PROGRAM ActuationSystems
VAR
fbMainJibCylinderHyd : ValveControlledCylinder;
fbKnuckleJibCylinderHyd : ValveControlledCylinder;
fbKingRotationCylinderHyd : ValveControlledCylinder;
//HydraulicCylinder
fbMainJibCylinderMech : CylinderMech;
fbKnuckleJibCylinderMech : CylinderMech;
fbkingRotationCylinderMech : CylinderMech;

fbHPU : HPU;
END_VAR

fbHPU(
);

//Hyd Model for MainJibCylinder (CONNECTED TO UNREAL)
fbMainJibCylinderHyd(
	uDcvEnable := Inputs.uDcvEnableMainJib,
	uDcv := Inputs.uDcvMainJib,	
	ReturnPressure := G_ActuationSystems.ReturnPressure,
	SupplyPressure := G_ActuationSystems.SupplyPressure,
	par := Param.pMainJibCylinder,
	xPiston := FromUnreal.MainJibPistPosition,
	vPiston := FromUnreal.MainJibPistVelocity,
	F_Hydraulic => ToUnreal.MainJibPistForce
);
//Hyd Model for KnuckleJibCylinder
fbKnuckleJibCylinderHyd(
	uDcvEnable := Inputs.uDcvEnableKnuckleJib,
	uDcv := Inputs.uDcvKnuckleJib,	
	ReturnPressure := G_ActuationSystems.ReturnPressure,
	SupplyPressure := G_ActuationSystems.SupplyPressure,
	par := Param.pKnuckleJibCylinder,
	xPiston := fbKnuckleJibCylinderMech.PistonPosition,
	vPiston := fbKnuckleJibCylinderMech.PistonVelocity
);

//Temp Mechanical Model for MainJibCylinder
fbMainJibCylinderMech(
	F_Hydraulic := fbMainJibCylinderHyd.F_Hydraulic,
	param := Param.pMainJibCylinder,
	F_Piston => Work.FpistonMainJib
);	

fbKnuckleJibCylinderMech(
	F_Hydraulic := fbKnuckleJibCylinderHyd.F_Hydraulic,
	param := Param.pKnuckleJibCylinder,
	F_Piston => Work.FpistonKnuckleJib
);

END_PROGRAM

(* stored: Version 1.1.0.1, ProductVersion 3.1.4024.9
   POU ActuationSystems: Id {3cabdd9c-217f-443b-9923-404fabc5dbf5}, SpecialFunc None *)
